{attribute 'strict'}
{attribute 'to_string'}
TYPE MachineState_enum :
(
	MS_OFF		 	:= 0,
	MS_RESTARTING	:= 1,
	MS_RUNNING		:= 2,
	MS_CYCLESTOP	:= 3,
	MS_STOPPING		:= 4,
	MS_ERROR		:= 5
);
END_TYPE

(* stored: Version 1.1.0.1, ProductVersion 3.1.4026.8
   DUT MachineState_enum: Id {18b48550-1ade-0961-2747-2f4a90c789e8} *)
